Fanuc KAREL source: test_kd_tree.kl

PROGRAM test_kd_tree
%NOLOCKGROUP

%include systemlib.types.klt
%include systemvars.klt
%include binary_tree.c.klt

%include kd_tree.klt
define_kd_types(T_KDQUEUE,tstkd,REAL)

%include pathlib.klt
define_kd_types(T_QUEUE_PTH,tkdph,REAL)

VAR
  data : PATH nodedata = t_VECTOR
  pth : PATH nodedata = t_VEC_PATH

%include kunit.klh
%from systemlib.klh %import VEC2D
%from display.klh %import clear, show

--vector data kdtree
%class tstkd('kd_tree.klc', 'kd_tree.klh', 'default_kd_dist.klt')
define_kd_headers(tstkd)

--vector path data kd tree
%class tkdph('kd_tree.klc', 'kd_tree.klh', 'kd_vec_path.klt')
define_kd_headers(tkdph)

ROUTINE clear_data
  VAR
    i : INTEGER
    status : INTEGER
  BEGIN
    i = PATH_LEN(data)
    WHILE PATH_LEN(data) > 0 DO
		  DELETE_NODE(data,i,status)
      i = i - 1
	  ENDWHILE
  END clear_data

ROUTINE clear_path
  VAR
    i : INTEGER
    status : INTEGER
  BEGIN
    i = PATH_LEN(pth)
    WHILE PATH_LEN(pth) > 0 DO
		  DELETE_NODE(pth,i,status)
      i = i - 1
	  ENDWHILE
  END clear_path


--          (7,2)
--    (5,4)       (9,6)
-- (2,3) (4,7)  (8,1)
ROUTINE t_insert : BOOLEAN
  VAR
    i, status : INTEGER
    nde : t_VECTOR
    exp, act : ARRAY[6] OF VECTOR
  BEGIN
    clear_data

    APPEND_NODE(data, status) ; data[1].v = VEC2D(7,2) ;
    APPEND_NODE(data, status) ; data[2].v = VEC2D(5,4) ;
    APPEND_NODE(data, status) ; data[3].v = VEC2D(9,6) ;
    APPEND_NODE(data, status) ; data[4].v = VEC2D(4,7) ;
    APPEND_NODE(data, status) ; data[5].v = VEC2D(8,1) ;
    APPEND_NODE(data, status) ; data[6].v = VEC2D(2,3) ;

    tstkd__create(data, (ZEROPOS(1)))

    tstkd__new_generator(PRE_ORDER)
    FOR i=1 TO ARRAY_LEN(act) DO
      nde = tstkd__next
      act[i] = nde.v
    ENDFOR

    exp[1] = VEC2D(7,2) ; exp[2] = VEC2D(5,4) ; exp[3] = VEC2D(2,3) ;
    exp[4] = VEC2D(4,7) ; exp[5] = VEC2D(9,6) ; exp[6] = VEC2D(8,1) ;


    RETURN(kunit_eq_arv(exp, act, 0.05) )

   END t_insert

--            (35,45)
--      (5,25)      (70,70)
-- (10,12) (30,40)     (50,30)

--               (50,50)
--        (25,40)      (51,75)
--   (10,30) (35,90)     (70,70)
-- (1,10)             (55,1) (60,80)
ROUTINE t_insert2 : BOOLEAN
  VAR
    i, status : INTEGER
    nde : t_VECTOR
    exp, act : ARRAY[9] OF VECTOR
  BEGIN
    clear_data

    APPEND_NODE(data, status) ; data[1].v = VEC2D(51,75) ;
    APPEND_NODE(data, status) ; data[2].v = VEC2D(25,40) ;
    APPEND_NODE(data, status) ; data[3].v = VEC2D(70,70) ;
    APPEND_NODE(data, status) ; data[4].v = VEC2D(10,30) ;
    APPEND_NODE(data, status) ; data[5].v = VEC2D(35,90) ;
    APPEND_NODE(data, status) ; data[6].v = VEC2D(55,1) ;
    APPEND_NODE(data, status) ; data[7].v = VEC2D(60,80) ;
    APPEND_NODE(data, status) ; data[8].v = VEC2D(1,10) ;
    APPEND_NODE(data, status) ; data[9].v = VEC2D(50,50) ;

    tstkd__create(data, (ZEROPOS(1)))

    tstkd__new_generator(PRE_ORDER)
    FOR i=1 TO ARRAY_LEN(act) DO
      nde = tstkd__next
      act[i] = nde.v
    ENDFOR

    exp[1] = VEC2D(50,50) ; exp[2] = VEC2D(25,40) ; exp[3] = VEC2D(10,30) ;
    exp[4] = VEC2D(1,10) ; exp[5] = VEC2D(35,90) ; exp[6] = VEC2D(51,75) ;
    exp[7] = VEC2D(70,70) ; exp[8] = VEC2D(55,1) ; exp[9] = VEC2D(60,80) ;

    RETURN(kunit_eq_arv(exp, act, 0.05) )

   END t_insert2

--               (50,50)
--        (25,40)      (51,75)
--   (10,30) (35,90)     (70,70)
-- (1,10)             (55,1) (60,80)
ROUTINE t_min : BOOLEAN
  VAR
    mn_x, mn_y : t_VECTOR
    act1, exp1 : VECTOR
    act2, exp2 : VECTOR
    status : INTEGER
  BEGIN
    clear_data

    APPEND_NODE(data, status) ; data[1].v = VEC2D(51,75) ;
    APPEND_NODE(data, status) ; data[2].v = VEC2D(25,40) ;
    APPEND_NODE(data, status) ; data[3].v = VEC2D(70,70) ;
    APPEND_NODE(data, status) ; data[4].v = VEC2D(10,30) ;
    APPEND_NODE(data, status) ; data[5].v = VEC2D(35,90) ;
    APPEND_NODE(data, status) ; data[6].v = VEC2D(55,1) ;
    APPEND_NODE(data, status) ; data[7].v = VEC2D(60,80) ;
    APPEND_NODE(data, status) ; data[8].v = VEC2D(1,10) ;
    APPEND_NODE(data, status) ; data[9].v = VEC2D(50,50) ;

    tstkd__create(data, (ZEROPOS(1)))

    mn_x = tstkd__findmin(1)
    act1 = mn_x.v
    exp1 = VEC2D(1,10)

    mn_y = tstkd__findmin(2)
    act2 = mn_y.v
    exp2 = VEC2D(55,1)

    RETURN(kunit_eq_vec(exp1,act1) AND kunit_eq_vec(exp2,act2) )

  END t_min

--               (50,50)
--        (25,40)      (51,75)
--   (10,30) (35,90)     (70,70)
-- (1,10)             (55,1) (60,80)
ROUTINE t_max : BOOLEAN
  VAR
    mx_x, mx_y : t_VECTOR
    act1, exp1 : VECTOR
    act2, exp2 : VECTOR
    status : INTEGER
  BEGIN
    clear_data

    APPEND_NODE(data, status) ; data[1].v = VEC2D(51,75) ;
    APPEND_NODE(data, status) ; data[2].v = VEC2D(25,40) ;
    APPEND_NODE(data, status) ; data[3].v = VEC2D(70,70) ;
    APPEND_NODE(data, status) ; data[4].v = VEC2D(10,30) ;
    APPEND_NODE(data, status) ; data[5].v = VEC2D(35,90) ;
    APPEND_NODE(data, status) ; data[6].v = VEC2D(55,1) ;
    APPEND_NODE(data, status) ; data[7].v = VEC2D(60,80) ;
    APPEND_NODE(data, status) ; data[8].v = VEC2D(1,10) ;
    APPEND_NODE(data, status) ; data[9].v = VEC2D(50,50) ;

    tstkd__create(data, (ZEROPOS(1)))

    mx_x = tstkd__findmax(1)
    act1 = mx_x.v
    exp1 = VEC2D(70,70)

    mx_y = tstkd__findmax(2)
    act2 = mx_y.v
    exp2 = VEC2D(35,90)

    RETURN(kunit_eq_vec(exp1,act1) AND kunit_eq_vec(exp2,act2) )

  END t_max

ROUTINE t_NN : BOOLEAN
  VAR
    point : t_VECTOR
    status : INTEGER
    act1, exp1 : ARRAY[2] OF VECTOR
    act2, exp2 : ARRAY[3] OF VECTOR
  BEGIN
    clear_data

    APPEND_NODE(data, status) ; data[1].v = VEC2D(51,75) ;
    APPEND_NODE(data, status) ; data[2].v = VEC2D(25,40) ;
    APPEND_NODE(data, status) ; data[3].v = VEC2D(70,70) ;
    APPEND_NODE(data, status) ; data[4].v = VEC2D(10,30) ;
    APPEND_NODE(data, status) ; data[5].v = VEC2D(35,90) ;
    APPEND_NODE(data, status) ; data[6].v = VEC2D(55,1) ;
    APPEND_NODE(data, status) ; data[7].v = VEC2D(60,80) ;
    APPEND_NODE(data, status) ; data[8].v = VEC2D(1,10) ;
    APPEND_NODE(data, status) ; data[9].v = VEC2D(50,50) ;

    tstkd__create(data, (ZEROPOS(1)))

    point.v = VEC2D(10,10)
    tstkd__kth_nearest_neighbors(point, 2)
    tstkd__get_query_arr(act1)

    exp1[1] = VEC2D(1,10) ; exp1[2] = VEC2D(10,30)

    point.v = VEC2D(80,30)
    tstkd__kth_nearest_neighbors(point, 3)
    tstkd__get_query_arr(act2)

    exp2[1] = VEC2D(50,50) ; exp2[2] = VEC2D(55,1) ;
    exp2[3] = VEC2D(70,70)

    RETURN(kunit_eq_arv(exp1, act1, 0.05) AND kunit_eq_arv(exp2, act2, 0.05) )

  END t_NN

ROUTINE t_NN_Brute : BOOLEAN
  VAR
    point : t_VECTOR
    status : INTEGER
    act1, exp1 : ARRAY[2] OF VECTOR
    act2, exp2 : ARRAY[3] OF VECTOR
  BEGIN
    clear_data

    APPEND_NODE(data, status) ; data[1].v = VEC2D(51,75) ;
    APPEND_NODE(data, status) ; data[2].v = VEC2D(25,40) ;
    APPEND_NODE(data, status) ; data[3].v = VEC2D(70,70) ;
    APPEND_NODE(data, status) ; data[4].v = VEC2D(10,30) ;
    APPEND_NODE(data, status) ; data[5].v = VEC2D(35,90) ;
    APPEND_NODE(data, status) ; data[6].v = VEC2D(55,1) ;
    APPEND_NODE(data, status) ; data[7].v = VEC2D(60,80) ;
    APPEND_NODE(data, status) ; data[8].v = VEC2D(1,10) ;
    APPEND_NODE(data, status) ; data[9].v = VEC2D(50,50) ;

    point.v = VEC2D(10,10)
    tstkd__kNN_brute_force(point, 2, data)
    tstkd__get_query_arr(act1)

    exp1[1] = VEC2D(1,10) ; exp1[2] = VEC2D(10,30)

    point.v = VEC2D(80,30)
    tstkd__kNN_brute_force(point, 3, data)
    tstkd__get_query_arr(act2)

    exp2[1] = VEC2D(50,50) ; exp2[2] = VEC2D(55,1) ;
    exp2[3] = VEC2D(70,70)

    RETURN(kunit_eq_arv(exp1, act1, 0.05) AND kunit_eq_arv(exp2, act2, 0.05) )

  END t_NN_Brute

ROUTINE t_NNR : BOOLEAN
  VAR
    point : t_VECTOR
    radius : REAL
    status : INTEGER
    act, exp : ARRAY[3] OF VECTOR
  BEGIN
    clear_data

    APPEND_NODE(data, status) ; data[1].v = VEC2D(51,75) ;
    APPEND_NODE(data, status) ; data[2].v = VEC2D(25,40) ;
    APPEND_NODE(data, status) ; data[3].v = VEC2D(70,70) ;
    APPEND_NODE(data, status) ; data[4].v = VEC2D(10,30) ;
    APPEND_NODE(data, status) ; data[5].v = VEC2D(35,90) ;
    APPEND_NODE(data, status) ; data[6].v = VEC2D(55,1) ;
    APPEND_NODE(data, status) ; data[7].v = VEC2D(60,80) ;
    APPEND_NODE(data, status) ; data[8].v = VEC2D(1,10) ;
    APPEND_NODE(data, status) ; data[9].v = VEC2D(50,50) ;

    tstkd__create(data, (ZEROPOS(1)))

    point.v = VEC2D(60,70)
    radius = 20
    tstkd__radius_nearest_neighbors(point, radius)
    tstkd__get_query_arr(act)

    exp[1] = VEC2D(70,70) ; exp[2] = VEC2D(60,80) ;
    exp[3] = VEC2D(51,75)

    RETURN(kunit_eq_arv(exp, act, 0.05) )

  END t_NNR

ROUTINE t_NNR_brute : BOOLEAN
  VAR
    point : t_VECTOR
    radius : REAL
    status : INTEGER
    act, exp : ARRAY[3] OF VECTOR
  BEGIN
    clear_data

    APPEND_NODE(data, status) ; data[1].v = VEC2D(51,75) ;
    APPEND_NODE(data, status) ; data[2].v = VEC2D(25,40) ;
    APPEND_NODE(data, status) ; data[3].v = VEC2D(70,70) ;
    APPEND_NODE(data, status) ; data[4].v = VEC2D(10,30) ;
    APPEND_NODE(data, status) ; data[5].v = VEC2D(35,90) ;
    APPEND_NODE(data, status) ; data[6].v = VEC2D(55,1) ;
    APPEND_NODE(data, status) ; data[7].v = VEC2D(60,80) ;
    APPEND_NODE(data, status) ; data[8].v = VEC2D(1,10) ;
    APPEND_NODE(data, status) ; data[9].v = VEC2D(50,50) ;

    point.v = VEC2D(60,70)
    radius = 20
    tstkd__rNN_brute_force(point, radius, data)
    tstkd__get_query_arr(act)

    exp[1] = VEC2D(70,70) ; exp[2] = VEC2D(60,80) ;
    exp[3] = VEC2D(51,75)

    RETURN(kunit_eq_arv(exp, act, 0.05) )

  END t_NNR_brute

--                  (25,40)
--        (51,75)             (50,50)
--    (10,30) (60,80)     (55,1)  (70,70)
-- (35,90)             (1,10)
ROUTINE t_conv : BOOLEAN
  VAR
    i, status : INTEGER
    nde : t_VECTOR
    exp, act : ARRAY[9] OF VECTOR
  BEGIN
    clear_data

    APPEND_NODE(data, status) ; data[1].v = VEC2D(51,75) ;
    APPEND_NODE(data, status) ; data[2].v = VEC2D(25,40) ;
    APPEND_NODE(data, status) ; data[3].v = VEC2D(70,70) ;
    APPEND_NODE(data, status) ; data[4].v = VEC2D(10,30) ;
    APPEND_NODE(data, status) ; data[5].v = VEC2D(35,90) ;
    APPEND_NODE(data, status) ; data[6].v = VEC2D(55,1) ;
    APPEND_NODE(data, status) ; data[7].v = VEC2D(60,80) ;
    APPEND_NODE(data, status) ; data[8].v = VEC2D(1,10) ;
    APPEND_NODE(data, status) ; data[9].v = VEC2D(50,50) ;

    tstkd__create(data, POS(0,0,0,0,0,-45,(ZEROPOS(1).Config_data) ))

    tstkd__new_generator(PRE_ORDER)
    FOR i=1 TO ARRAY_LEN(act) DO
      nde = tstkd__next
      act[i] = nde.v
    ENDFOR

    exp[1] = VEC2D(25,40) ; exp[2] = VEC2D(51,75) ; exp[3] = VEC2D(10,30) ;
    exp[4] = VEC2D(35,90) ; exp[5] = VEC2D(60,80) ; exp[6] = VEC2D(50,50) ;
    exp[7] = VEC2D(55,1) ; exp[8] = VEC2D(1,10) ; exp[9] = VEC2D(70,70) ;

    RETURN(kunit_eq_arv(exp, act, 0.05) )

  END t_conv

ROUTINE t_hexagon : BOOLEAN
  VAR
    i, status : INTEGER
    act,exp : ARRAY[4] OF VECTOR
  BEGIN
    clear_data

    --hexagon raster lines
    APPEND_NODE(data, status) ; data[1].v = VEC2D(44.721, 122.472) ;
    APPEND_NODE(data, status) ; data[2].v = VEC2D(44.721, 177.528) ;
    APPEND_NODE(data, status) ; data[3].v = VEC2D(64.721, 94.945) ;
    APPEND_NODE(data, status) ; data[4].v = VEC2D(64.721, 205.055) ;
    APPEND_NODE(data, status) ; data[5].v = VEC2D(84.721, 67.417) ;
    APPEND_NODE(data, status) ; data[6].v = VEC2D(84.721, 232.583) ;
    APPEND_NODE(data, status) ; data[7].v = VEC2D(104.721, 39.889) ;
    APPEND_NODE(data, status) ; data[8].v = VEC2D(104.721, 260.111) ;
    APPEND_NODE(data, status) ; data[9].v = VEC2D(124.721, 35.218) ;
    APPEND_NODE(data, status) ; data[10].v = VEC2D(124.721, 264.782) ;
    APPEND_NODE(data, status) ; data[11].v = VEC2D(144.721, 41.716) ;
    APPEND_NODE(data, status) ; data[12].v = VEC2D(144.721, 258.284) ;
    APPEND_NODE(data, status) ; data[13].v = VEC2D(164.721, 48.215) ;
    APPEND_NODE(data, status) ; data[14].v = VEC2D(164.721, 251.785) ;
    APPEND_NODE(data, status) ; data[15].v = VEC2D(184.721, 54.713) ;
    APPEND_NODE(data, status) ; data[16].v = VEC2D(184.721, 245.287) ;
    APPEND_NODE(data, status) ; data[17].v = VEC2D(204.721, 61.212) ;
    APPEND_NODE(data, status) ; data[18].v = VEC2D(204.721, 238.788) ;
    APPEND_NODE(data, status) ; data[19].v = VEC2D(224.721, 67.710) ;
    APPEND_NODE(data, status) ; data[20].v = VEC2D(224.721, 232.290) ;
    APPEND_NODE(data, status) ; data[21].v = VEC2D(244.721, 74.208) ;
    APPEND_NODE(data, status) ; data[22].v = VEC2D(244.721, 225.792) ;

    -- raster direction VEC2D(-1,0)
    tstkd__create(data, POS(0,0,0,0,0,90,(ZEROPOS(1).Config_data) ))

    tstkd__kth_nearest_neighbors(data[13], 4)
    tstkd__get_query_arr(act)

    exp[1] = VEC2D(184.72,54.71) ; exp[2] = VEC2D(144.72,41.72) ; exp[3] = VEC2D(124.72,35.22) ;
    exp[4] = VEC2D(204.72,61.21) ;

    RETURN(kunit_eq_arv(exp, act, 0.05) )

  END t_hexagon


ROUTINE t_path : BOOLEAN
  VAR
    i, status : INTEGER
    nde : t_VEC_PATH
    act, exp : ARRAY[5] OF VECTOR
  BEGIN
    clear_path
    -- L
    APPEND_NODE(pth, status) ; pth[1].v = VEC2D(-4,4) ;       pth[1].code = PTH_MOVETO ;  pth[1].polygon = 1
    APPEND_NODE(pth, status) ; pth[2].v = VEC2D(-4,0) ;       pth[2].code = PTH_LINETO ;  pth[2].polygon = 1
    APPEND_NODE(pth, status) ; pth[3].v = VEC2D(-0.5,0) ;     pth[3].code = PTH_LINETO ;  pth[3].polygon = 1
    APPEND_NODE(pth, status) ; pth[4].v = VEC2D(-0.5,1) ;     pth[4].code = PTH_LINETO ;  pth[4].polygon = 1
    APPEND_NODE(pth, status) ; pth[5].v = VEC2D(-2.5,1) ;     pth[5].code = PTH_LINETO ;  pth[5].polygon = 1
    APPEND_NODE(pth, status) ; pth[6].v = VEC2D(-2.5,4) ;     pth[6].code = PTH_LINETO ;  pth[6].polygon = 1
    APPEND_NODE(pth, status) ; pth[7].v = VEC2D(-4,4) ;       pth[7].code = PTH_CLOSE ;   pth[7].polygon = 1
    -- O
    APPEND_NODE(pth, status) ; pth[8].v = VEC2D(2,4) ;        pth[8].code = PTH_MOVETO ;  pth[8].polygon = 2
    APPEND_NODE(pth, status) ; pth[9].v = VEC2D(0,2) ;        pth[9].code = PTH_CURVE3 ;  pth[9].polygon = 2
    APPEND_NODE(pth, status) ; pth[10].v = VEC2D(2,0) ;       pth[10].code = PTH_CURVE3 ; pth[10].polygon = 2
    APPEND_NODE(pth, status) ; pth[11].v = VEC2D(4,2) ;       pth[11].code = PTH_CURVE3 ; pth[11].polygon = 2
    APPEND_NODE(pth, status) ; pth[12].v = VEC2D(2,4) ;       pth[12].code = PTH_CLOSE ;  pth[12].polygon = 2
    APPEND_NODE(pth, status) ; pth[13].v = VEC2D(1,2) ;       pth[13].code = PTH_MOVETO ; pth[13].polygon = 2
    APPEND_NODE(pth, status) ; pth[14].v = VEC2D(2,1) ;       pth[14].code = PTH_CURVE3 ; pth[14].polygon = 2
    APPEND_NODE(pth, status) ; pth[15].v = VEC2D(3,2) ;       pth[15].code = PTH_CURVE3 ; pth[15].polygon = 2
    APPEND_NODE(pth, status) ; pth[16].v = VEC2D(2,3) ;       pth[16].code = PTH_CURVE3 ; pth[16].polygon = 2
    APPEND_NODE(pth, status) ; pth[17].v = VEC2D(1,2) ;       pth[17].code = PTH_CLOSE ;  pth[17].polygon = 2
    -- G
    APPEND_NODE(pth, status) ; pth[18].v = VEC2D(-2,-1.5) ;   pth[18].code = PTH_MOVETO ; pth[18].polygon = 3
    APPEND_NODE(pth, status) ; pth[19].v = VEC2D(-2,-2.4) ;   pth[19].code = PTH_LINETO ; pth[19].polygon = 3
    APPEND_NODE(pth, status) ; pth[20].v = VEC2D(-1,-2.4) ;   pth[20].code = PTH_LINETO ; pth[20].polygon = 3
    APPEND_NODE(pth, status) ; pth[21].v = VEC2D(-2,-3) ;     pth[21].code = PTH_CURVE3 ; pth[21].polygon = 3
    APPEND_NODE(pth, status) ; pth[22].v = VEC2D(-3,-2) ;     pth[22].code = PTH_CURVE3 ; pth[22].polygon = 3
    APPEND_NODE(pth, status) ; pth[23].v = VEC2D(-2,-1) ;     pth[23].code = PTH_CURVE3 ; pth[23].polygon = 3
    APPEND_NODE(pth, status) ; pth[24].v = VEC2D(-1.4,-1.2) ; pth[24].code = PTH_CURVE3 ; pth[24].polygon = 3
    APPEND_NODE(pth, status) ; pth[25].v = VEC2D(-0.6,-0.6) ; pth[25].code = PTH_LINETO ; pth[25].polygon = 3
    APPEND_NODE(pth, status) ; pth[26].v = VEC2D(-2,0) ;      pth[26].code = PTH_CURVE3 ; pth[26].polygon = 3
    APPEND_NODE(pth, status) ; pth[27].v = VEC2D(-4,-2) ;     pth[27].code = PTH_CURVE3 ; pth[27].polygon = 3
    APPEND_NODE(pth, status) ; pth[28].v = VEC2D(-2,-4) ;     pth[28].code = PTH_CURVE3 ; pth[28].polygon = 3
    APPEND_NODE(pth, status) ; pth[29].v = VEC2D(0,-1.5) ;    pth[29].code = PTH_CURVE3 ; pth[29].polygon = 3
    APPEND_NODE(pth, status) ; pth[30].v = VEC2D(-2,-1.5) ;   pth[30].code = PTH_CLOSE ;  pth[30].polygon = 3
    -- O
    APPEND_NODE(pth, status) ; pth[31].v = VEC2D(0,-2) ;      pth[31].code = PTH_MOVETO ; pth[31].polygon = 4
    APPEND_NODE(pth, status) ; pth[32].v = VEC2D(2,-4) ;      pth[32].code = PTH_CURVE3 ; pth[32].polygon = 4
    APPEND_NODE(pth, status) ; pth[33].v = VEC2D(4,-2) ;      pth[33].code = PTH_CURVE3 ; pth[33].polygon = 4
    APPEND_NODE(pth, status) ; pth[34].v = VEC2D(2,0) ;       pth[34].code = PTH_CURVE3 ; pth[34].polygon = 4
    APPEND_NODE(pth, status) ; pth[35].v = VEC2D(0,-2) ;      pth[35].code = PTH_CLOSE ;  pth[35].polygon = 4
    APPEND_NODE(pth, status) ; pth[36].v = VEC2D(2,-1) ;      pth[36].code = PTH_MOVETO ; pth[36].polygon = 4
    APPEND_NODE(pth, status) ; pth[37].v = VEC2D(1,-2) ;      pth[37].code = PTH_CURVE3 ; pth[37].polygon = 4
    APPEND_NODE(pth, status) ; pth[38].v = VEC2D(2,-3) ;      pth[38].code = PTH_CURVE3 ; pth[38].polygon = 4
    APPEND_NODE(pth, status) ; pth[39].v = VEC2D(3,-2) ;      pth[39].code = PTH_CURVE3 ; pth[39].polygon = 4
    APPEND_NODE(pth, status) ; pth[40].v = VEC2D(2,-1) ;      pth[40].code = PTH_CLOSE ;  pth[40].polygon = 4
    -- circle
    APPEND_NODE(pth, status) ; pth[41].v = VEC2D(0,6) ;       pth[41].code = PTH_MOVETO ; pth[41].polygon = 5
    APPEND_NODE(pth, status) ; pth[42].v = VEC2D(-6,0) ;      pth[42].code = PTH_CURVE3 ; pth[42].polygon = 5
    APPEND_NODE(pth, status) ; pth[43].v = VEC2D(0,-6) ;      pth[43].code = PTH_CURVE3 ; pth[43].polygon = 5
    APPEND_NODE(pth, status) ; pth[44].v = VEC2D(6,0) ;       pth[44].code = PTH_CURVE3 ; pth[44].polygon = 5
    APPEND_NODE(pth, status) ; pth[45].v = VEC2D(0,6) ;       pth[45].code = PTH_CLOSE ;  pth[45].polygon = 5

    tkdph__create_filtered(pth, (ZEROPOS(1)))

    tkdph__kth_nearest_neighbors(pth[35], 5)
    tkdph__get_query_arr(act)

    exp[1] = VEC2D(-2,-1.5) ; exp[2] = VEC2D(2,-1) ; exp[3] = VEC2D(1,2) ;
    exp[4] = VEC2D(2,4) ; exp[5] = VEC2D(-4,4) ;

    RETURN(kunit_eq_arv(exp, act, 0.05) )
  END t_path

BEGIN
  -- total asserts 15
  kunit_test('test kd tree', t_insert) --assert 1
  kunit_test('test kd tree 2', t_insert2) --assert 1
  kunit_test('min nodes', t_min) --assert 2
  kunit_test('max nodes', t_max) --assert 2
  kunit_test('kth nearest neighbor', t_NN) --assert 2
  kunit_test('kth nearest neighbor brute force', t_NN_Brute) --assert 2
  kunit_test('nearest neighbor radius', t_NNR) --assert 1
  kunit_test('nearest neighbor radius brute force', t_NNR_Brute) --assert 1
  kunit_test('frame convolution test', t_conv) --asserts 1
  kunit_test('hexagon nearest neighbors', t_hexagon) --asserts 1
  kunit_test('vector path kd tree', t_path) --asserts 1
  kunit_done


  --destructor
  tstkd__clear
END test_kd_tree
